PROGRAM SendCommands 
VAR
	
END_VAR

//socketconnect
VAR_INPUT
        sSrvNetId       : T_AmsNetId := '192.168.10.15';
        sRemoteHost     : STRING(15);
        nRemotePort     : UDINT;
        bExecute                : BOOL;
        tTimeout                : TIME := T#45s;(*!!!*)
END_VAR

VAR_OUTPUT
        bBusy           : BOOL;
        bError          : BOOL;
        nErrId          : UDINT;
        hSocket         : T_HSOCKET;
END_VAR



//sockettsend
VAR_INPUT
        sSrvNetId2    : T_AmsNetId := '192.168.10.15';    
        hSocket2	      : T_HSOCKET;          
        cbLen           : UDINT;                        
        pSrc            : DWORD;                        
        bExecute2                : BOOL;                 
        tTimeout2               : TIME := T#5S;         
END_VAR

VAR_OUTPUT
        bBusy2           : BOOL;
        bError2         : BOOL;
        nErrId2          : UDINT;
END_VAR




sRemoteHost := '192.168.10.10';
nRemotePort := 7142;



IF gvl1.socketconnectknop = TRUE THEN
	bExecute := TRUE;
hSocket := hSocket2;

END_IF

IF GVL1.socketsendknop = TRUE THEN
	hSocket := hSocket2;
	pSrc := Beamer_Projectorscherm.BeamerAAN;
	bExecute2 := TRUE;
END_IF

END_PROGRAM

(* stored: Version 1.1.0.1, ProductVersion 3.1.4022.9
   POU SendCommands: Id {8a796357-d5f5-4bfd-9c3d-8a0926e64f1e}, SpecialFunc None *)
